GLOBALCONSTANTS virtuals (* Global constants *)
  (* Standard: 61499-1 *)
  (* Version 1.0, 2025-05-16, mow *)
  VAR_GLOBAL CONSTANT
    local : WSTRING := "xquery[127.0.0.1:1984; BaSys_PalletSystem_Model; test; test]";
  END_VAR
END_GLOBALCONSTANTS
